// SIMATIC S7-200 project (STEP 7-Micro/WIN), CPU 224 REL 01.11

SYMBOL_TABLE USER1
ON_OFF           I0.0
X1               Q0.0
V1               Q0.1
D1               Q0.2
X2               Q0.3
V2               Q0.4
D2               Q0.5
END_SYMBOL_TABLE

ORGANIZATION_BLOCK MAIN:OB1
TITLE=PROGRAM COMMENTS
BEGIN
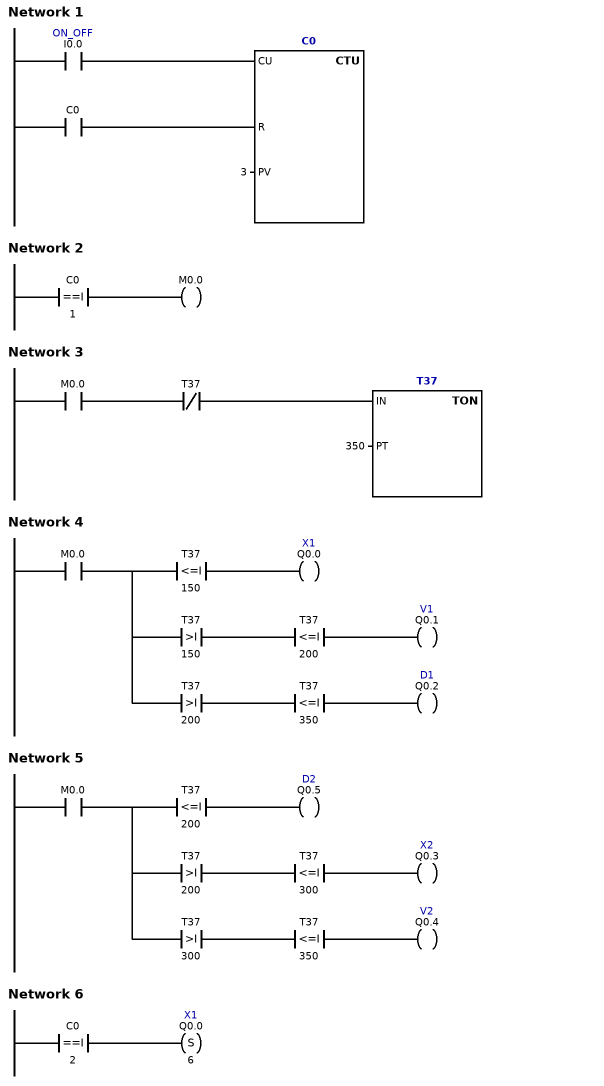
Network 1
LD     ON_OFF:I0.0
LD     C0
CTU    C0, 3
Network 2
LDW=   C0, 1
=      M0.0
Network 3
LD     M0.0
AN     T37
TON    T37, 350
Network 4
LD     M0.0
LPS
AW<=   T37, 150
=      X1:Q0.0
LRD
AW>    T37, 150
AW<=   T37, 200
=      V1:Q0.1
LPP
AW>    T37, 200
AW<=   T37, 350
=      D1:Q0.2
Network 5
LD     M0.0
LPS
AW<=   T37, 200
=      D2:Q0.5
LRD
AW>    T37, 200
AW<=   T37, 300
=      X2:Q0.3
LPP
AW>    T37, 300
AW<=   T37, 350
=      V2:Q0.4
Network 6
LDW=   C0, 2
S      X1:Q0.0, 6
END_ORGANIZATION_BLOCK
